TEXTLIST TL_TempSensType
  0 = 'NoSensor'
  1 = 'TC_B'
  2 = 'TC_E'
  3 = 'TC_J'
  4 = 'TC_K'
  5 = 'TC_L'
  6 = 'TC_N'
  7 = 'TC_R'
  8 = 'TC_S'
  9 = 'TC_T'
  10 = 'TC_U'
  100 = 'PT_100'
  101 = 'NI_100'
  102 = 'NI_120'
  103 = 'PT_200'
  104 = 'PT_500'
  105 = 'PT_1000'
  106 = 'NI_1000'
  10000 = 'Customized'
   = ''
END_TEXTLIST

(* stored: Version 1.1.0.1, ProductVersion 3.1.4018.5
   TextList TL_TempSensType: Id {9c42961a-d0bf-4eba-8702-b063261b9955} *)
